TYPE ServicesTimingParts :
STRUCT
	///I/O modules
	io: ServicesTimingIO;
	///Info acquired by serial link
	serialInfo: ServicesTimingSerialInfo;
END_STRUCT
END_TYPE

(* stored: Version 1.1.0.1, ProductVersion 3.1.4019.2
   DUT ServicesTimingParts: Id {d87db6e9-5a27-4f95-bded-01693ce1db67} *)
